Staubli VAL3: listredraw.pgx

public program listredraw(num pFirst (dimensions=1))
begin
  //
  // Staubli Copyright 2003 06 20
  //
  call listframe(sTitle,nTopX,nTopY,nBottomX,nBottomY)
  call listupdate(pFirst)
end
